FUNCTION_BLOCK MapBOOL2INT
  (* Standard: 61499-2 *)
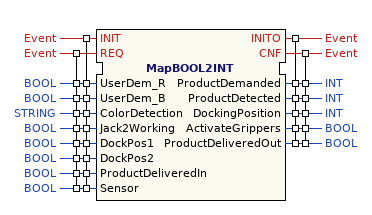
  EVENT_INPUT
    INIT WITH UserDem_R, UserDem_B, ColorDetection, Jack2Working, DockPos1, DockPos2, ProductDeliveredIn, Sensor;
    REQ WITH UserDem_R, UserDem_B, ColorDetection, Jack2Working, DockPos1, DockPos2, ProductDeliveredIn, Sensor;
  END_EVENT
  EVENT_OUTPUT
    INITO WITH ProductDemanded, ProductDetected, DockingPosition, ActivateGrippers, ProductDeliveredOut;
    CNF WITH ProductDemanded, ProductDetected, DockingPosition, ActivateGrippers, ProductDeliveredOut;
  END_EVENT
  VAR_INPUT
    UserDem_R : BOOL;
    UserDem_B : BOOL;
    ColorDetection : STRING;
    Jack2Working : BOOL;
    DockPos1 : BOOL;
    DockPos2 : BOOL;
    ProductDeliveredIn : BOOL;
    Sensor : BOOL;
  END_VAR
  VAR_OUTPUT
    ProductDemanded : INT;
    ProductDetected : INT;
    DockingPosition : INT;
    ActivateGrippers : BOOL;
    ProductDeliveredOut : BOOL;
  END_VAR
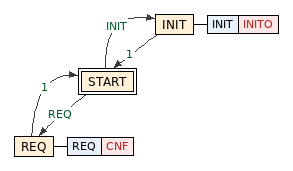
  EC_STATES
    START;
    INIT : INIT -> INITO;
    REQ : REQ -> CNF;
  END_STATES
  EC_TRANSITIONS
    START TO INIT := INIT;
    INIT TO START := 1;
    START TO REQ := REQ;
    REQ TO START := 1;
  END_TRANSITIONS
  ALGORITHM INIT IN ST:

  END_ALGORITHM
  ALGORITHM REQ IN ST:

  END_ALGORITHM
END_FUNCTION_BLOCK
